FUNCTION_BLOCK SetSafetySimulationVisitor IMPLEMENTS I_ComponentVisitor
VAR
	SafetyComponent : I_SafetyBase;
	InfoData		: ST_SafetyStateDiag;
	_Simulated		: BOOL;
END_VAR

PROPERTY Diag : UINT
SET
InfoData.Diag := Diag;
END_SET
END_PROPERTY

PROPERTY Simulated : BOOL
GET
Simulated := _Simulated;
END_GET
SET
_Simulated := Simulated;
END_SET
END_PROPERTY

PROPERTY State : USINT
SET
InfoData.State := State;
END_SET
END_PROPERTY

METHOD VisitComponent
VAR_INPUT
	Component : I_Component;
END_VAR
IF __QUERYINTERFACE(Component, SafetyComponent) THEN
	SafetyComponent.Simulated := _Simulated;
	SafetyComponent.SimulateSafetyDiag(InfoData.Diag);
	SafetyComponent.SimulateSafetyState(InfoData.State);
END_IF
END_METHOD

END_FUNCTION_BLOCK

(* stored: Version 1.1.0.1, ProductVersion 3.1.4026.18
   POU SetSafetySimulationVisitor: Id {79102bb4-a0f7-4ee5-9427-b177ab4334f8}, SpecialFunc None
   Property Diag: Id {7a1ddad5-8f39-4d1e-87da-b5052b1d418d}
   Set Set: Id {8166e58e-686c-460f-a3e1-5eb1bb404148}
   Property Simulated: Id {a9e80197-9312-4336-a27a-75b318350a40}
   Get Get: Id {2e4a40fa-d007-422b-a194-2e0cd694ccbc}
   Set Set: Id {2b44dbcf-0407-4121-af7a-a86c14213ed3}
   Property State: Id {02f3e22b-889d-46c9-ac40-8fa5db0d3242}
   Set Set: Id {3218036a-fcc6-4da0-8d8f-5933bdc1724f}
   Method VisitComponent: Id {7c119b81-f287-4983-a57c-5d070e320c65} *)
